// Mitsubishi GX Developer project: Lab4   PLC: FX1S

PROGRAM MAIN
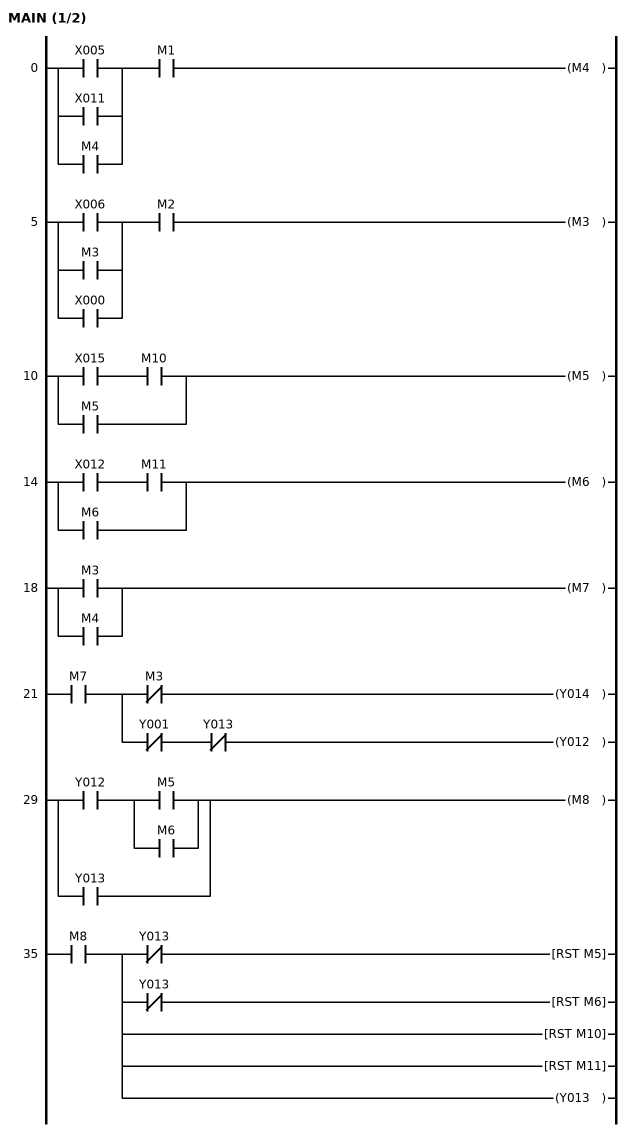
0     LD      X005
      OR      X011
      OR      M4
      AND     M1
      OUT     M4
5     LD      X006
      OR      M3
      OR      X000
      AND     M2
      OUT     M3
10    LD      X015
      AND     M10
      OR      M5
      OUT     M5
14    LD      X012
      AND     M11
      OR      M6
      OUT     M6
18    LD      M3
      OR      M4
      OUT     M7
21    LD      M7
      MPS
      ANI     M3
      OUT     Y014
      MPP
      ANI     Y001
      ANI     Y013
      OUT     Y012
29    LD      Y012
      LD      M5
      OR      M6
      ANB
      OR      Y013
      OUT     M8
35    LD      M8
      MPS
      ANI     Y013
      RST     M5
      MRD
      ANI     Y013
      RST     M6
      MPP
      RST     M10
      RST     M11
      OUT     Y013
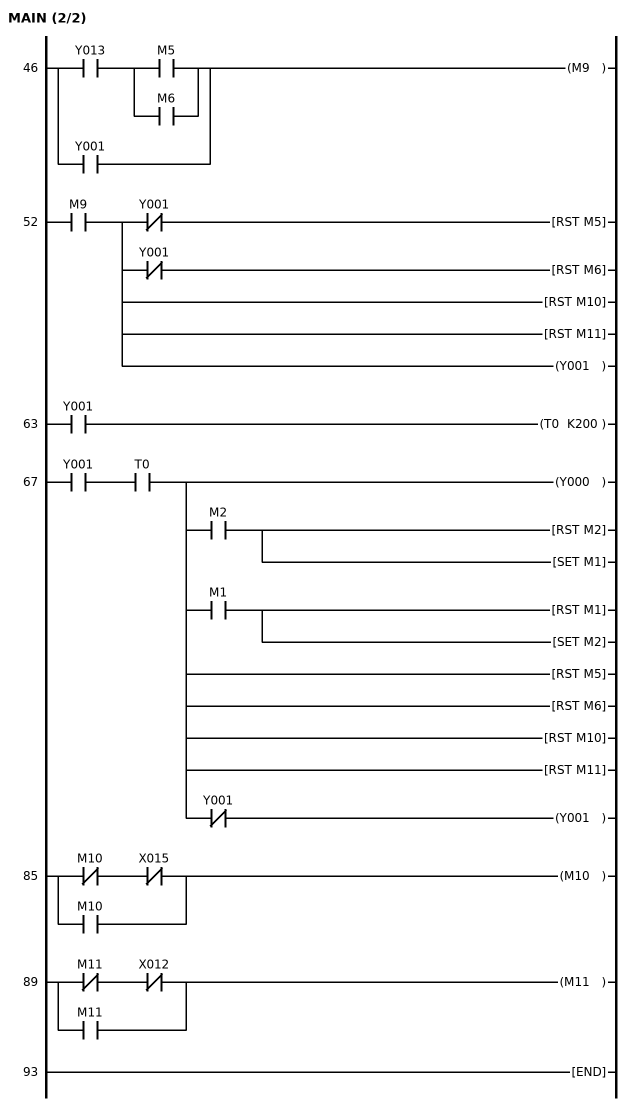
46    LD      Y013
      LD      M5
      OR      M6
      ANB
      OR      Y001
      OUT     M9
52    LD      M9
      MPS
      ANI     Y001
      RST     M5
      MRD
      ANI     Y001
      RST     M6
      MPP
      RST     M10
      RST     M11
      OUT     Y001
63    LD      Y001
      OUT     T0 K200
67    LD      Y001
      AND     T0
      OUT     Y000
      MPS
      AND     M2
      RST     M2
      SET     M1
      MRD
      AND     M1
      RST     M1
      SET     M2
      MPP
      RST     M5
      RST     M6
      RST     M10
      RST     M11
      ANI     Y001
      OUT     Y001
85    LDI     M10
      ANI     X015
      OR      M10
      OUT     M10
89    LDI     M11
      ANI     X012
      OR      M11
      OUT     M11
93    END
END_PROGRAM
